FUNCTION_BLOCK Test (* Composite Function Block Type *)
  (* Standard: 61499-2 *)
  (* Version 0.0, 7/14/2016, Andrei, nxtControl GmbH, template *)
  PACKAGE Main;
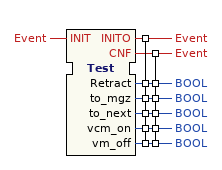
  EVENT_INPUT
    INIT; (* Initialization Request *)
  END_EVENT
  EVENT_OUTPUT
    INITO WITH Retract, to_mgz, to_next, vcm_on, vm_off; (* Initialization Confirm *)
    CNF WITH Retract, to_mgz, to_next, vcm_on, vm_off; (* Execution Confirmation *)
  END_EVENT
  VAR_OUTPUT
    Retract : BOOL; (* Output event qualifier *)
    to_mgz : BOOL;
    to_next : BOOL;
    vcm_on : BOOL;
    vm_off : BOOL;
  END_VAR
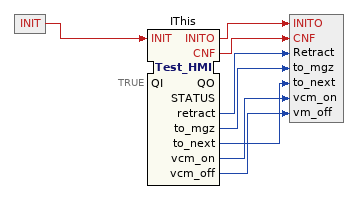
  FBS
    IThis : Test_HMI(QI := TRUE);
  END_FBS
  EVENT_CONNECTIONS
    INIT TO IThis.INIT;
    IThis.INITO TO INITO;
    IThis.CNF TO CNF;
  END_CONNECTIONS
  DATA_CONNECTIONS
    IThis.retract TO Retract;
    IThis.to_mgz TO to_mgz;
    IThis.to_next TO to_next;
    IThis.vcm_on TO vcm_on;
    IThis.vcm_off TO vm_off;
  END_CONNECTIONS
END_FUNCTION_BLOCK
